// TIA Portal V19 export
DATA_BLOCK "HMI"   // DB50
// stored: Access Published, MemoryReserve 0
   VAR
      PLCDateTime : DTL;
      ProjectInfo : "ProjectInfo";
      AreaGen : Struct
         Status : "StatusArea";
         Pb_SafetyRstAll : Bool;
         Sgn_SafetyRstAll : Bool;
         Pb_LampTest : Bool;
      END_STRUCT;
   END_VAR
BEGIN
END_DATA_BLOCK
